FUNCTION_BLOCK SequenceTransfer
VAR_INPUT	
    Execute:BOOL;
	Next: INT;
	Hold: BOOL;
END_VAR
VAR_OUTPUT
	Last: INT;
	Now: INT;
END_VAR
VAR_IN_OUT
END_VAR

IF Execute AND NOT Hold THEN
   Last:=Now;
   Now:=Next;
   Execute:=FALSE;
END_IF

END_FUNCTION_BLOCK

(* stored: Version 1.1.0.1, ProductVersion 3.1.4022.16
   POU SequenceTransfer: Id {15e3dac5-1803-4bd2-a45f-a13fe28c8e65}, SpecialFunc None *)
